FUNCTION_BLOCK TRANTEST (* Test of Eventless Transitions *)
  (* Standard: 61499-1 *)
  (* Version 0.0, 2006-03-20, JHC, Holobloc Inc *)
  (* Compiler header: package fb.rt.test; *)
  (* Compiler Java Sun JDK 1.5.0 *)
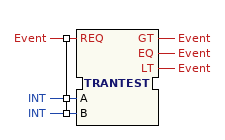
  EVENT_INPUT
    REQ WITH A, B; (* Normal Execution Request *)
  END_EVENT
  EVENT_OUTPUT
    GT; (* A > B *)
    EQ; (* A = B *)
    LT; (* A < B *)
  END_EVENT
  VAR_INPUT
    A : INT;
    B : INT;
  END_VAR
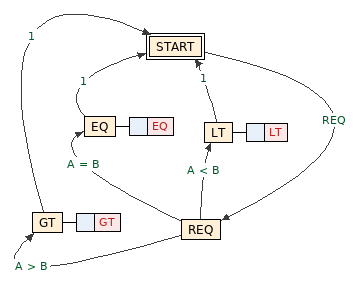
  EC_STATES
    START; (* Initial State *)
    REQ; (* Normal execution *)
    GT : -> GT;
    EQ : -> EQ;
    LT : -> LT;
  END_STATES
  EC_TRANSITIONS
    START TO REQ := REQ;
    REQ TO GT := A > B;
    REQ TO EQ := A = B;
    REQ TO LT := A < B;
    GT TO START := 1;
    EQ TO START := 1;
    LT TO START := 1;
  END_TRANSITIONS
END_FUNCTION_BLOCK
